FUNCTION F_sigmoid : LREAL
VAR_INPUT
	x : LREAL;
END_VAR

IF x > 1E2 THEN
	F_sigmoid := 1;
ELSIF x < -1E2 THEN
	F_sigmoid := 0;
ELSE
	F_sigmoid := 1 / (1 + EXP(-x));
END_IF

END_FUNCTION

(* stored: Version 1.1.0.1, ProductVersion 3.1.4024.12
   POU F_sigmoid: Id {06514012-fa58-4a56-a5df-a893c7a5bf78}, SpecialFunc None *)
